TYPE (* A Template for a Data Type *)
  (* Version 1.0, 2026-04-10, hyperion *)
  PACKAGE forte::eclipse4diac::io::ethercat;
  ECSlaveConfig : STRUCT
    Alias : UINT;
    Position : UINT;
    VendorId : UDINT;
    ProductCode : UDINT;
  END_STRUCT;
END_TYPE
